FUNCTION_BLOCK FB_4PVICI_EPS 
VAR_INPUT
    iAddress : INT;
END_VAR
VAR_OUTPUT
    bAllPortsLocked : BOOL;
    bExternalLock : BOOL;
END_VAR
VAR_IN_OUT
    aPortEPS : ARRAY [*] OF E_VICI_PORT_EPS; // EPS for each port.
END_VAR
VAR
	
	{attribute 'pytmc' := '
        pv: ''
        io: io
    '}
    fbNporValveEPS : FB_ViciValveEPS;
    iNumPorts : INT := 4;

    {attribute 'pytmc' := '
        pv: SampleNames
        io: io
     '}
    stSampleNames : ST_4PViciValveSampleNames;	

END_VAR

fbNporValveEPS(iAddress := iAddress,
    iNumOfPorts := iNumPorts,
	aPortEPS := aPortEPS,
	bAllPortsLocked => bAllPortsLocked,
	bExternalLock => bExternalLock);

END_FUNCTION_BLOCK

(* stored: Version 1.1.0.1, ProductVersion 3.1.4024.12
   POU FB_4PVICI_EPS: Id {89dd5800-3edc-4db3-a7b8-40f2bc027efe}, SpecialFunc None *)
